// TwinCAT 3 PLC project project
// ProgramVersion: 3.1.4023.0
// libraries:
//   Tc2_Standard, * (Beckhoff Automation GmbH)
//   Tc2_System, * (Beckhoff Automation GmbH)
//   Tc3_Module, * (Beckhoff Automation GmbH)
// project tree:
//   / PlcTask.TcTTO (not stored)
//   POUs/ MAIN.TcPOU, POU_1.TcPOU
// real-time tasks:
//   TASK PlcTask: cycle T#10ms, priority 20, ADS port 350

// ---- POUs/MAIN.TcPOU
PROGRAM MAIN
VAR
END_VAR

POU_1();

END_PROGRAM

// ---- POUs/POU_1.TcPOU
PROGRAM POU_1
VAR
	
	objectDetected : BOOL := FALSE;

	blackObject : BOOL := FALSE;	
	redObject : BOOL := FALSE;
	
	motorOn : BOOL := FALSE;
	actuatorMove : BOOL := FALSE;
	
	objectSorted : BOOL := FALSE;
	
	startTimer : BOOL := FALSE;
	TON_0 : TON;	

END_VAR

END_PROGRAM
